{attribute 'qualified_only'}
{attribute 'strict'}
TYPE E_LaudaParameterReadState :
(
	READY := 0,
	ACTUAL_TEMPERATURE_SETPOINT,
	BAH_OUTFLOW_TEMP,
	PUMP_STAGE,
	READ_ENABLE_STATE,
	OIL_LEVEL,
	FAULT_DIAGNOSIS,
	DONE
);
END_TYPE

(* stored: Version 1.1.0.1, ProductVersion 3.1.4024.13
   DUT E_LaudaParameterReadState: Id {f98eae1c-c5c5-4744-b6cd-541bfbf682e3} *)
